// TIA Portal V17 export
// export: Created 2026-04-13T11:12:43.5468084Z, ExportSetting WithDefaults, DisplayName Totally Integrated Automation Portal, DisplayVersion V17 Update 4, DisplayName TIA Portal Openness, DisplayVersion V17 Update 4, DisplayName TIA Portal Version Control Interface, DisplayVersion V17, DisplayName SINAMICS Startdrive Advanced, DisplayVersion V17, DisplayName SINAMICS Startdrive G130, G150, S120, S150, SINAMICS MV, S210, DisplayVersion V17, DisplayName SINAMICS Startdrive G110M, G120, G120C, G120D, G120P, G115D, DisplayVersion V17, DisplayName STEP 7 Professional, DisplayVersion V17 Update 4, DisplayName STEP 7 Safety, DisplayVersion V17, DisplayName WinCC Professional, DisplayVersion V17 Update 4
FUNCTION_BLOCK "30-加热控制"   // FB17, SCL
{ S7_Optimized_Access := 'TRUE' }
VERSION : 0.1
// stored: AutoNumber true, IsIECCheckEnabled false, IsRetainMemResEnabled false, MemoryReserve 100, SetENOAutomatically false, UDAEnableTagReadback false
   VAR_INPUT
      条件1 : Real;
   END_VAR
   VAR_IN_OUT
      模式设定 : Real;
      加热控制按钮 : Bool;
      电力调整器信号 : Bool;
      电力调整器报警 : Bool;
      机械温报警信号 : Bool;
      循环风机反馈 : Real;
      循环风机 : Bool;
      加热输出 : Bool;
      AO : Int;
      安全停机 : Bool;
   END_VAR
BEGIN

   //手动控制--------------------------------------------------------------------------------------------------------------
   IF #模式设定 = 2.0 THEN
       //预热器加热手动控制
       IF #加热控制按钮
           AND #电力调整器报警 = FALSE AND #机械温报警信号 = FALSE AND #循环风机反馈 > 20 AND #循环风机 THEN
           #加热输出 := TRUE;

       ELSE

           #加热输出 := FALSE;

       END_IF;
   END_IF;
   IF #模式设定 = 2.0  THEN
       //预热器加热手动控制
       IF NOT #加热控制按钮 THEN


           #加热输出 := FALSE;

       END_IF;
   END_IF;

   //自动模式
   IF #加热输出 THEN
       #AO := -256;
   END_IF;


   IF NOT #加热输出 THEN
       #AO := 0;
   END_IF;
   IF #电力调整器信号 THEN
       #电力调整器报警 := TRUE;
   ELSE


       #电力调整器报警 := FALSE;
   END_IF;

   IF
       #模式设定 = 1 AND (#电力调整器报警 OR #机械温报警信号) THEN

       #安全停机 := 1;
   END_IF;
END_FUNCTION_BLOCK
